  PROC DrawPart12()
    MoveL Offs(pOrigin,191.45,110.32,6.00),vTravel,z5,tPen\WObj:=wPaper;
    MoveL Offs(pOrigin,191.45,110.32,0.00),v60,z0,tPen\WObj:=wPaper;
    MoveL Offs(pOrigin,191.50,109.88,0.00),v40,z0,tPen\WObj:=wPaper;
    MoveL Offs(pOrigin,193.40,108.07,0.00),v40,fine,tPen\WObj:=wPaper;
    MoveL Offs(pOrigin,193.40,108.07,6.00),v60,z5,tPen\WObj:=wPaper;
    MoveL Offs(pOrigin,194.60,106.72,6.00),vTravel,z5,tPen\WObj:=wPaper;
    MoveL Offs(pOrigin,194.60,106.72,0.00),v60,z0,tPen\WObj:=wPaper;
    MoveL Offs(pOrigin,195.65,107.03,0.00),v40,z0,tPen\WObj:=wPaper;
    MoveL Offs(pOrigin,195.65,107.03,0.00),v40,z0,tPen\WObj:=wPaper;
    MoveL Offs(pOrigin,197.00,108.68,0.00),v40,z0,tPen\WObj:=wPaper;
    MoveL Offs(pOrigin,197.00,108.68,0.00),v40,z0,tPen\WObj:=wPaper;
    MoveL Offs(pOrigin,197.45,111.07,0.00),v40,z0,tPen\WObj:=wPaper;
    MoveL Offs(pOrigin,197.45,111.07,0.00),v40,z0,tPen\WObj:=wPaper;
    MoveL Offs(pOrigin,198.05,112.28,0.00),v40,z0,tPen\WObj:=wPaper;
    MoveL Offs(pOrigin,198.05,112.28,0.00),v40,z0,tPen\WObj:=wPaper;
    MoveL Offs(pOrigin,199.10,113.78,0.00),v40,z0,tPen\WObj:=wPaper;
    MoveL Offs(pOrigin,199.10,115.72,0.00),v40,z0,tPen\WObj:=wPaper;
    MoveL Offs(pOrigin,198.05,118.28,0.00),v40,z0,tPen\WObj:=wPaper;
    MoveL Offs(pOrigin,191.30,125.03,0.00),v40,z0,tPen\WObj:=wPaper;
    MoveL Offs(pOrigin,188.75,125.03,0.00),v40,fine,tPen\WObj:=wPaper;
    MoveL Offs(pOrigin,188.75,125.03,6.00),v60,z5,tPen\WObj:=wPaper;
    MoveL Offs(pOrigin,190.25,121.43,6.00),vTravel,z5,tPen\WObj:=wPaper;
    MoveL Offs(pOrigin,190.25,121.43,0.00),v60,z0,tPen\WObj:=wPaper;
    MoveL Offs(pOrigin,190.70,121.12,0.00),v40,z0,tPen\WObj:=wPaper;
    MoveL Offs(pOrigin,190.85,119.93,0.00),v40,z0,tPen\WObj:=wPaper;
    MoveL Offs(pOrigin,190.85,119.93,0.00),v40,z0,tPen\WObj:=wPaper;
    MoveL Offs(pOrigin,197.15,113.93,0.00),v40,z0,tPen\WObj:=wPaper;
    MoveL Offs(pOrigin,197.15,113.93,0.00),v40,z0,tPen\WObj:=wPaper;
    MoveL Offs(pOrigin,197.35,112.88,0.00),v40,z0,tPen\WObj:=wPaper;
    MoveL Offs(pOrigin,198.05,112.28,0.00),v40,fine,tPen\WObj:=wPaper;
    MoveL Offs(pOrigin,198.05,112.28,6.00),v60,z5,tPen\WObj:=wPaper;
    MoveL Offs(pOrigin,197.15,113.93,6.00),vTravel,z5,tPen\WObj:=wPaper;
    MoveL Offs(pOrigin,197.15,113.93,0.00),v60,z0,tPen\WObj:=wPaper;
    MoveL Offs(pOrigin,198.50,114.82,0.00),v40,fine,tPen\WObj:=wPaper;
    MoveL Offs(pOrigin,198.50,114.82,6.00),v60,z5,tPen\WObj:=wPaper;
    MoveL Offs(pOrigin,203.45,112.57,6.00),vTravel,z5,tPen\WObj:=wPaper;
    MoveL Offs(pOrigin,203.45,112.57,0.00),v60,z0,tPen\WObj:=wPaper;
    MoveL Offs(pOrigin,204.80,116.93,0.00),v40,fine,tPen\WObj:=wPaper;
    MoveL Offs(pOrigin,204.80,116.93,6.00),v60,z5,tPen\WObj:=wPaper;
    MoveL Offs(pOrigin,205.55,118.28,6.00),vTravel,z5,tPen\WObj:=wPaper;
    MoveL Offs(pOrigin,205.55,118.28,0.00),v60,z0,tPen\WObj:=wPaper;
    MoveL Offs(pOrigin,209.15,114.43,0.00),v40,z0,tPen\WObj:=wPaper;
    MoveL Offs(pOrigin,210.65,113.62,0.00),v40,z0,tPen\WObj:=wPaper;
    MoveL Offs(pOrigin,210.65,113.62,0.00),v40,z0,tPen\WObj:=wPaper;
    MoveL Offs(pOrigin,210.65,113.93,0.00),v40,z0,tPen\WObj:=wPaper;
    MoveL Offs(pOrigin,210.95,113.93,0.00),v40,z0,tPen\WObj:=wPaper;
    MoveL Offs(pOrigin,210.95,113.62,0.00),v40,z0,tPen\WObj:=wPaper;
    MoveL Offs(pOrigin,210.95,113.62,0.00),v40,z0,tPen\WObj:=wPaper;
    MoveL Offs(pOrigin,215.00,109.43,0.00),v40,z0,tPen\WObj:=wPaper;
    MoveL Offs(pOrigin,215.00,109.43,0.00),v40,z0,tPen\WObj:=wPaper;
    MoveL Offs(pOrigin,215.75,110.03,0.00),v40,z0,tPen\WObj:=wPaper;
    MoveL Offs(pOrigin,215.75,110.03,0.00),v40,z0,tPen\WObj:=wPaper;
    MoveL Offs(pOrigin,216.50,110.78,0.00),v40,z0,tPen\WObj:=wPaper;
    MoveL Offs(pOrigin,217.55,115.72,0.00),v40,z0,tPen\WObj:=wPaper;
    MoveL Offs(pOrigin,216.50,120.53,0.00),v40,z0,tPen\WObj:=wPaper;
    MoveL Offs(pOrigin,215.75,121.28,0.00),v40,z0,tPen\WObj:=wPaper;
    MoveL Offs(pOrigin,215.75,121.28,0.00),v40,z0,tPen\WObj:=wPaper;
    MoveL Offs(pOrigin,210.95,116.32,0.00),v40,z0,tPen\WObj:=wPaper;
    MoveL Offs(pOrigin,210.35,115.57,0.00),v40,z0,tPen\WObj:=wPaper;
    MoveL Offs(pOrigin,215.75,110.03,0.00),v40,z0,tPen\WObj:=wPaper;
    MoveL Offs(pOrigin,215.00,109.43,0.00),v40,z0,tPen\WObj:=wPaper;
    MoveL Offs(pOrigin,214.65,108.38,0.00),v40,z0,tPen\WObj:=wPaper;
    MoveL Offs(pOrigin,213.80,108.03,0.00),v40,z0,tPen\WObj:=wPaper;
    MoveL Offs(pOrigin,213.35,107.22,0.00),v40,z0,tPen\WObj:=wPaper;
    MoveL Offs(pOrigin,212.80,107.03,0.00),v40,z0,tPen\WObj:=wPaper;
    MoveL Offs(pOrigin,212.35,104.62,0.00),v40,z0,tPen\WObj:=wPaper;
    MoveL Offs(pOrigin,211.15,102.97,0.00),v40,z0,tPen\WObj:=wPaper;
    MoveL Offs(pOrigin,210.50,100.12,0.00),v40,z0,tPen\WObj:=wPaper;
    MoveL Offs(pOrigin,210.50,100.12,0.00),v40,z0,tPen\WObj:=wPaper;
    MoveL Offs(pOrigin,213.65,97.03,0.00),v40,z0,tPen\WObj:=wPaper;
    MoveL Offs(pOrigin,221.15,95.18,0.00),v40,z0,tPen\WObj:=wPaper;
    MoveL Offs(pOrigin,226.55,93.22,0.00),v40,fine,tPen\WObj:=wPaper;
    MoveL Offs(pOrigin,226.55,93.22,6.00),v60,z5,tPen\WObj:=wPaper;
    MoveL Offs(pOrigin,217.25,86.18,6.00),vTravel,z5,tPen\WObj:=wPaper;
    MoveL Offs(pOrigin,217.25,86.18,0.00),v60,z0,tPen\WObj:=wPaper;
    MoveL Offs(pOrigin,214.85,88.62,0.00),v40,z0,tPen\WObj:=wPaper;
    MoveL Offs(pOrigin,213.05,88.72,0.00),v40,z0,tPen\WObj:=wPaper;
    MoveL Offs(pOrigin,213.05,88.72,0.00),v40,z0,tPen\WObj:=wPaper;
    MoveL Offs(pOrigin,212.30,87.68,0.00),v40,z0,tPen\WObj:=wPaper;
    MoveL Offs(pOrigin,212.50,86.78,0.00),v40,z0,tPen\WObj:=wPaper;
    MoveL Offs(pOrigin,213.05,86.22,0.00),v40,z0,tPen\WObj:=wPaper;
    MoveL Offs(pOrigin,217.25,86.18,0.00),v40,z0,tPen\WObj:=wPaper;
    MoveL Offs(pOrigin,217.25,86.18,0.00),v40,z0,tPen\WObj:=wPaper;
    MoveL Offs(pOrigin,219.95,83.32,0.00),v40,z0,tPen\WObj:=wPaper;
    MoveL Offs(pOrigin,219.95,83.32,0.00),v40,z0,tPen\WObj:=wPaper;
    MoveL Offs(pOrigin,217.70,81.07,0.00),v40,z0,tPen\WObj:=wPaper;
    MoveL Offs(pOrigin,216.80,80.93,0.00),v40,z0,tPen\WObj:=wPaper;
    MoveL Offs(pOrigin,216.80,80.93,0.00),v40,z0,tPen\WObj:=wPaper;
    MoveL Offs(pOrigin,215.95,80.03,0.00),v40,z0,tPen\WObj:=wPaper;
    MoveL Offs(pOrigin,215.95,79.43,0.00),v40,z0,tPen\WObj:=wPaper;
    MoveL Offs(pOrigin,220.25,75.32,0.00),v40,z0,tPen\WObj:=wPaper;
    MoveL Offs(pOrigin,220.85,75.07,0.00),v40,z0,tPen\WObj:=wPaper;
    MoveL Offs(pOrigin,225.80,75.07,0.00),v40,z0,tPen\WObj:=wPaper;
    MoveL Offs(pOrigin,225.80,75.07,0.00),v40,z0,tPen\WObj:=wPaper;
    MoveL Offs(pOrigin,225.20,70.43,0.00),v40,z0,tPen\WObj:=wPaper;
    MoveL Offs(pOrigin,224.75,69.68,0.00),v40,z0,tPen\WObj:=wPaper;
    MoveL Offs(pOrigin,224.75,69.68,0.00),v40,z0,tPen\WObj:=wPaper;
    MoveL Offs(pOrigin,224.30,68.03,0.00),v40,z0,tPen\WObj:=wPaper;
    MoveL Offs(pOrigin,222.80,67.07,0.00),v40,z0,tPen\WObj:=wPaper;
    MoveL Offs(pOrigin,221.00,64.43,0.00),v40,z0,tPen\WObj:=wPaper;
    MoveL Offs(pOrigin,220.10,63.97,0.00),v40,z0,tPen\WObj:=wPaper;
    MoveL Offs(pOrigin,220.10,63.97,0.00),v40,z0,tPen\WObj:=wPaper;
    MoveL Offs(pOrigin,214.60,69.38,0.00),v40,z0,tPen\WObj:=wPaper;
    MoveL Offs(pOrigin,214.55,69.82,0.00),v40,z0,tPen\WObj:=wPaper;
    MoveL Offs(pOrigin,214.55,69.82,0.00),v40,z0,tPen\WObj:=wPaper;
    MoveL Offs(pOrigin,215.00,70.88,0.00),v40,z0,tPen\WObj:=wPaper;
    MoveL Offs(pOrigin,214.55,69.82,0.00),v40,z0,tPen\WObj:=wPaper;
    MoveL Offs(pOrigin,212.75,71.47,0.00),v40,fine,tPen\WObj:=wPaper;
    MoveL Offs(pOrigin,212.75,71.47,6.00),v60,z5,tPen\WObj:=wPaper;
    MoveL Offs(pOrigin,210.80,70.57,6.00),vTravel,z5,tPen\WObj:=wPaper;
    MoveL Offs(pOrigin,210.80,70.57,0.00),v60,z0,tPen\WObj:=wPaper;
    MoveL Offs(pOrigin,211.85,71.43,0.00),v40,z0,tPen\WObj:=wPaper;
    MoveL Offs(pOrigin,213.20,71.93,0.00),v40,z0,tPen\WObj:=wPaper;
    MoveL Offs(pOrigin,214.25,73.88,0.00),v40,z0,tPen\WObj:=wPaper;
    MoveL Offs(pOrigin,214.25,73.88,0.00),v40,z0,tPen\WObj:=wPaper;
    MoveL Offs(pOrigin,214.60,75.53,0.00),v40,z0,tPen\WObj:=wPaper;
    MoveL Offs(pOrigin,215.15,76.28,0.00),v40,z0,tPen\WObj:=wPaper;
    MoveL Offs(pOrigin,215.15,76.28,0.00),v40,z0,tPen\WObj:=wPaper;
    MoveL Offs(pOrigin,215.45,78.38,0.00),v40,z0,tPen\WObj:=wPaper;
    MoveL Offs(pOrigin,215.45,78.38,0.00),v40,z0,tPen\WObj:=wPaper;
  ENDPROC

  PROC DrawPart13()
    MoveL Offs(pOrigin,215.90,79.28,0.00),v40,fine,tPen\WObj:=wPaper;
    MoveL Offs(pOrigin,215.90,79.28,6.00),v60,z5,tPen\WObj:=wPaper;
    MoveL Offs(pOrigin,216.35,80.78,6.00),vTravel,z5,tPen\WObj:=wPaper;
    MoveL Offs(pOrigin,216.35,80.78,0.00),v60,z0,tPen\WObj:=wPaper;
    MoveL Offs(pOrigin,214.40,80.93,0.00),v40,z0,tPen\WObj:=wPaper;
    MoveL Offs(pOrigin,212.00,81.68,0.00),v40,z0,tPen\WObj:=wPaper;
    MoveL Offs(pOrigin,208.85,81.68,0.00),v40,z0,tPen\WObj:=wPaper;
    MoveL Offs(pOrigin,207.35,82.18,0.00),v40,z0,tPen\WObj:=wPaper;
    MoveL Offs(pOrigin,206.00,83.62,0.00),v40,z0,tPen\WObj:=wPaper;
    MoveL Offs(pOrigin,206.30,85.43,0.00),v40,z0,tPen\WObj:=wPaper;
    MoveL Offs(pOrigin,206.30,85.43,0.00),v40,z0,tPen\WObj:=wPaper;
    MoveL Offs(pOrigin,203.00,88.57,0.00),v40,z0,tPen\WObj:=wPaper;
    MoveL Offs(pOrigin,202.85,89.18,0.00),v40,z0,tPen\WObj:=wPaper;
    MoveL Offs(pOrigin,202.85,89.18,0.00),v40,z0,tPen\WObj:=wPaper;
    MoveL Offs(pOrigin,203.60,89.93,0.00),v40,z0,tPen\WObj:=wPaper;
    MoveL Offs(pOrigin,203.60,89.93,0.00),v40,z0,tPen\WObj:=wPaper;
    MoveL Offs(pOrigin,202.85,89.18,0.00),v40,z0,tPen\WObj:=wPaper;
    MoveL Offs(pOrigin,202.85,89.18,0.00),v40,z0,tPen\WObj:=wPaper;
    MoveL Offs(pOrigin,202.25,89.93,0.00),v40,fine,tPen\WObj:=wPaper;
    MoveL Offs(pOrigin,202.25,89.93,6.00),v60,z5,tPen\WObj:=wPaper;
    MoveL Offs(pOrigin,203.60,89.93,6.00),vTravel,z5,tPen\WObj:=wPaper;
    MoveL Offs(pOrigin,203.60,89.93,0.00),v60,z0,tPen\WObj:=wPaper;
    MoveL Offs(pOrigin,204.35,89.78,0.00),v40,z0,tPen\WObj:=wPaper;
    MoveL Offs(pOrigin,206.90,87.38,0.00),v40,z0,tPen\WObj:=wPaper;
    MoveL Offs(pOrigin,206.90,87.38,0.00),v40,z0,tPen\WObj:=wPaper;
    MoveL Offs(pOrigin,206.90,86.18,0.00),v40,z0,tPen\WObj:=wPaper;
    MoveL Offs(pOrigin,206.30,85.43,0.00),v40,fine,tPen\WObj:=wPaper;
    MoveL Offs(pOrigin,206.30,85.43,6.00),v60,z5,tPen\WObj:=wPaper;
    MoveL Offs(pOrigin,206.90,87.38,6.00),vTravel,z5,tPen\WObj:=wPaper;
    MoveL Offs(pOrigin,206.90,87.38,0.00),v60,z0,tPen\WObj:=wPaper;
    MoveL Offs(pOrigin,209.30,88.88,0.00),v40,z0,tPen\WObj:=wPaper;
    MoveL Offs(pOrigin,208.85,88.28,0.00),v40,z0,tPen\WObj:=wPaper;
    MoveL Offs(pOrigin,209.60,88.88,0.00),v40,z0,tPen\WObj:=wPaper;
    MoveL Offs(pOrigin,213.05,88.72,0.00),v40,z0,tPen\WObj:=wPaper;
    MoveL Offs(pOrigin,213.05,88.72,0.00),v40,z0,tPen\WObj:=wPaper;
    MoveL Offs(pOrigin,212.30,87.97,0.00),v40,fine,tPen\WObj:=wPaper;
    MoveL Offs(pOrigin,212.30,87.97,6.00),v60,z5,tPen\WObj:=wPaper;
    MoveL Offs(pOrigin,211.70,85.43,6.00),vTravel,z5,tPen\WObj:=wPaper;
    MoveL Offs(pOrigin,211.70,85.43,0.00),v60,z0,tPen\WObj:=wPaper;
    MoveL Offs(pOrigin,211.50,86.18,0.00),v40,z0,tPen\WObj:=wPaper;
    MoveL Offs(pOrigin,210.20,86.78,0.00),v40,z0,tPen\WObj:=wPaper;
    MoveL Offs(pOrigin,208.85,88.28,0.00),v40,fine,tPen\WObj:=wPaper;
    MoveL Offs(pOrigin,208.85,88.28,6.00),v60,z5,tPen\WObj:=wPaper;
    MoveL Offs(pOrigin,206.00,83.32,6.00),vTravel,z5,tPen\WObj:=wPaper;
    MoveL Offs(pOrigin,206.00,83.32,0.00),v60,z0,tPen\WObj:=wPaper;
    MoveL Offs(pOrigin,205.40,81.82,0.00),v40,z0,tPen\WObj:=wPaper;
    MoveL Offs(pOrigin,205.40,81.82,0.00),v40,z0,tPen\WObj:=wPaper;
    MoveL Offs(pOrigin,205.55,80.47,0.00),v40,z0,tPen\WObj:=wPaper;
    MoveL Offs(pOrigin,205.55,80.47,0.00),v40,z0,tPen\WObj:=wPaper;
    MoveL Offs(pOrigin,205.05,79.88,0.00),v40,z0,tPen\WObj:=wPaper;
    MoveL Offs(pOrigin,204.50,77.62,0.00),v40,z0,tPen\WObj:=wPaper;
    MoveL Offs(pOrigin,204.50,77.62,0.00),v40,z0,tPen\WObj:=wPaper;
    MoveL Offs(pOrigin,203.90,76.88,0.00),v40,z0,tPen\WObj:=wPaper;
    MoveL Offs(pOrigin,203.90,76.88,0.00),v40,z0,tPen\WObj:=wPaper;
    MoveL Offs(pOrigin,203.45,74.93,0.00),v40,z0,tPen\WObj:=wPaper;
    MoveL Offs(pOrigin,203.45,74.93,0.00),v40,z0,tPen\WObj:=wPaper;
    MoveL Offs(pOrigin,205.55,73.28,0.00),v40,z0,tPen\WObj:=wPaper;
    MoveL Offs(pOrigin,206.60,71.62,0.00),v40,z0,tPen\WObj:=wPaper;
    MoveL Offs(pOrigin,208.25,69.97,0.00),v40,z0,tPen\WObj:=wPaper;
    MoveL Offs(pOrigin,208.25,69.53,0.00),v40,z0,tPen\WObj:=wPaper;
    MoveL Offs(pOrigin,209.00,70.53,0.00),v40,z0,tPen\WObj:=wPaper;
    MoveL Offs(pOrigin,210.80,70.57,0.00),v40,z0,tPen\WObj:=wPaper;
    MoveL Offs(pOrigin,210.80,70.57,0.00),v40,z0,tPen\WObj:=wPaper;
    MoveL Offs(pOrigin,211.80,69.53,0.00),v40,z0,tPen\WObj:=wPaper;
    MoveL Offs(pOrigin,212.45,67.88,0.00),v40,z0,tPen\WObj:=wPaper;
    MoveL Offs(pOrigin,218.15,62.33,0.00),v40,z0,tPen\WObj:=wPaper;
    MoveL Offs(pOrigin,218.15,62.33,0.00),v40,z0,tPen\WObj:=wPaper;
    MoveL Offs(pOrigin,218.15,61.88,0.00),v40,z0,tPen\WObj:=wPaper;
    MoveL Offs(pOrigin,217.55,61.58,0.00),v40,z0,tPen\WObj:=wPaper;
    MoveL Offs(pOrigin,217.55,61.58,0.00),v40,z0,tPen\WObj:=wPaper;
    MoveL Offs(pOrigin,212.90,66.22,0.00),v40,z0,tPen\WObj:=wPaper;
    MoveL Offs(pOrigin,212.00,66.72,0.00),v40,z0,tPen\WObj:=wPaper;
    MoveL Offs(pOrigin,211.45,66.22,0.00),v40,z0,tPen\WObj:=wPaper;
    MoveL Offs(pOrigin,211.85,65.47,0.00),v40,z0,tPen\WObj:=wPaper;
    MoveL Offs(pOrigin,212.15,65.18,0.00),v40,z0,tPen\WObj:=wPaper;
    MoveL Offs(pOrigin,216.80,60.53,0.00),v40,z0,tPen\WObj:=wPaper;
    MoveL Offs(pOrigin,216.80,60.53,0.00),v40,z0,tPen\WObj:=wPaper;
    MoveL Offs(pOrigin,217.55,61.58,0.00),v40,z0,tPen\WObj:=wPaper;
    MoveL Offs(pOrigin,218.15,62.33,0.00),v40,z0,tPen\WObj:=wPaper;
    MoveL Offs(pOrigin,219.35,62.78,0.00),v40,z0,tPen\WObj:=wPaper;
    MoveL Offs(pOrigin,220.10,63.97,0.00),v40,fine,tPen\WObj:=wPaper;
    MoveL Offs(pOrigin,220.10,63.97,6.00),v60,z5,tPen\WObj:=wPaper;
    MoveL Offs(pOrigin,221.90,65.93,6.00),vTravel,z5,tPen\WObj:=wPaper;
    MoveL Offs(pOrigin,221.90,65.93,0.00),v60,z0,tPen\WObj:=wPaper;
    MoveL Offs(pOrigin,214.25,73.57,0.00),v40,z0,tPen\WObj:=wPaper;
    MoveL Offs(pOrigin,213.35,73.88,0.00),v40,z0,tPen\WObj:=wPaper;
    MoveL Offs(pOrigin,213.05,73.72,0.00),v40,z0,tPen\WObj:=wPaper;
    MoveL Offs(pOrigin,213.05,74.03,0.00),v40,z0,tPen\WObj:=wPaper;
    MoveL Offs(pOrigin,213.35,73.88,0.00),v40,z0,tPen\WObj:=wPaper;
    MoveL Offs(pOrigin,213.05,73.72,0.00),v40,z0,tPen\WObj:=wPaper;
    MoveL Offs(pOrigin,213.05,74.03,0.00),v40,z0,tPen\WObj:=wPaper;
    MoveL Offs(pOrigin,213.35,73.88,0.00),v40,fine,tPen\WObj:=wPaper;
    MoveL Offs(pOrigin,213.35,73.88,6.00),v60,z5,tPen\WObj:=wPaper;
    MoveL Offs(pOrigin,213.50,76.72,6.00),vTravel,z5,tPen\WObj:=wPaper;
    MoveL Offs(pOrigin,213.50,76.72,0.00),v60,z0,tPen\WObj:=wPaper;
    MoveL Offs(pOrigin,215.00,78.22,0.00),v40,z0,tPen\WObj:=wPaper;
    MoveL Offs(pOrigin,213.50,76.72,0.00),v40,fine,tPen\WObj:=wPaper;
    MoveL Offs(pOrigin,213.50,76.72,6.00),v60,z5,tPen\WObj:=wPaper;
    MoveL Offs(pOrigin,215.15,76.28,6.00),vTravel,z5,tPen\WObj:=wPaper;
    MoveL Offs(pOrigin,215.15,76.28,0.00),v60,z0,tPen\WObj:=wPaper;
    MoveL Offs(pOrigin,218.30,73.43,0.00),v40,z0,tPen\WObj:=wPaper;
    MoveL Offs(pOrigin,219.35,71.78,0.00),v40,z0,tPen\WObj:=wPaper;
    MoveL Offs(pOrigin,223.40,67.72,0.00),v40,fine,tPen\WObj:=wPaper;
    MoveL Offs(pOrigin,223.40,67.72,6.00),v60,z5,tPen\WObj:=wPaper;
    MoveL Offs(pOrigin,224.75,69.68,6.00),vTravel,z5,tPen\WObj:=wPaper;
    MoveL Offs(pOrigin,224.75,69.68,0.00),v60,z0,tPen\WObj:=wPaper;
    MoveL Offs(pOrigin,221.00,73.43,0.00),v40,z0,tPen\WObj:=wPaper;
    MoveL Offs(pOrigin,220.10,73.57,0.00),v40,z0,tPen\WObj:=wPaper;
    MoveL Offs(pOrigin,219.95,73.88,0.00),v40,z0,tPen\WObj:=wPaper;
    MoveL Offs(pOrigin,220.10,74.03,0.00),v40,z0,tPen\WObj:=wPaper;
    MoveL Offs(pOrigin,220.40,74.03,0.00),v40,z0,tPen\WObj:=wPaper;
    MoveL Offs(pOrigin,220.40,73.72,0.00),v40,z0,tPen\WObj:=wPaper;
    MoveL Offs(pOrigin,220.10,74.03,0.00),v40,z0,tPen\WObj:=wPaper;
    MoveL Offs(pOrigin,220.40,74.03,0.00),v40,z0,tPen\WObj:=wPaper;
    MoveL Offs(pOrigin,220.25,73.72,0.00),v40,z0,tPen\WObj:=wPaper;
    MoveL Offs(pOrigin,220.10,74.03,0.00),v40,fine,tPen\WObj:=wPaper;
    MoveL Offs(pOrigin,220.10,74.03,6.00),v60,z5,tPen\WObj:=wPaper;
    MoveL Offs(pOrigin,225.80,75.07,6.00),vTravel,z5,tPen\WObj:=wPaper;
    MoveL Offs(pOrigin,225.80,75.07,0.00),v60,z0,tPen\WObj:=wPaper;
    MoveL Offs(pOrigin,226.25,77.78,0.00),v40,z0,tPen\WObj:=wPaper;
  ENDPROC

  PROC DrawPart14()
    MoveL Offs(pOrigin,225.95,80.32,0.00),v40,z0,tPen\WObj:=wPaper;
    MoveL Offs(pOrigin,225.35,81.78,0.00),v40,z0,tPen\WObj:=wPaper;
    MoveL Offs(pOrigin,222.20,83.32,0.00),v40,z0,tPen\WObj:=wPaper;
    MoveL Offs(pOrigin,220.25,83.32,0.00),v40,z0,tPen\WObj:=wPaper;
    MoveL Offs(pOrigin,217.70,80.93,0.00),v40,fine,tPen\WObj:=wPaper;
    MoveL Offs(pOrigin,217.70,80.93,6.00),v60,z5,tPen\WObj:=wPaper;
    MoveL Offs(pOrigin,209.75,78.53,6.00),vTravel,z5,tPen\WObj:=wPaper;
    MoveL Offs(pOrigin,209.75,78.53,0.00),v60,z0,tPen\WObj:=wPaper;
    MoveL Offs(pOrigin,210.20,78.22,0.00),v40,z0,tPen\WObj:=wPaper;
    MoveL Offs(pOrigin,210.05,77.78,0.00),v40,z0,tPen\WObj:=wPaper;
    MoveL Offs(pOrigin,209.75,77.93,0.00),v40,fine,tPen\WObj:=wPaper;
    MoveL Offs(pOrigin,209.75,77.93,6.00),v60,z5,tPen\WObj:=wPaper;
    MoveL Offs(pOrigin,209.90,75.53,6.00),vTravel,z5,tPen\WObj:=wPaper;
    MoveL Offs(pOrigin,209.90,75.53,0.00),v60,z0,tPen\WObj:=wPaper;
    MoveL Offs(pOrigin,208.70,75.53,0.00),v40,z0,tPen\WObj:=wPaper;
    MoveL Offs(pOrigin,207.95,75.97,0.00),v40,fine,tPen\WObj:=wPaper;
    MoveL Offs(pOrigin,207.95,75.97,6.00),v60,z5,tPen\WObj:=wPaper;
    MoveL Offs(pOrigin,207.95,74.62,6.00),vTravel,z5,tPen\WObj:=wPaper;
    MoveL Offs(pOrigin,207.95,74.62,0.00),v60,z0,tPen\WObj:=wPaper;
    MoveL Offs(pOrigin,207.95,74.18,0.00),v40,z0,tPen\WObj:=wPaper;
    MoveL Offs(pOrigin,208.70,73.88,0.00),v40,z0,tPen\WObj:=wPaper;
    MoveL Offs(pOrigin,208.70,73.88,0.00),v40,z0,tPen\WObj:=wPaper;
    MoveL Offs(pOrigin,209.55,74.32,0.00),v40,z0,tPen\WObj:=wPaper;
    MoveL Offs(pOrigin,209.90,75.53,0.00),v40,fine,tPen\WObj:=wPaper;
    MoveL Offs(pOrigin,209.90,75.53,6.00),v60,z5,tPen\WObj:=wPaper;
    MoveL Offs(pOrigin,209.60,74.18,6.00),vTravel,z5,tPen\WObj:=wPaper;
    MoveL Offs(pOrigin,209.60,74.18,0.00),v60,z0,tPen\WObj:=wPaper;
    MoveL Offs(pOrigin,209.45,73.57,0.00),v40,z0,tPen\WObj:=wPaper;
    MoveL Offs(pOrigin,208.85,73.57,0.00),v40,z0,tPen\WObj:=wPaper;
    MoveL Offs(pOrigin,208.70,73.88,0.00),v40,z0,tPen\WObj:=wPaper;
    MoveL Offs(pOrigin,208.70,73.57,0.00),v40,z0,tPen\WObj:=wPaper;
    MoveL Offs(pOrigin,208.85,70.57,0.00),v40,fine,tPen\WObj:=wPaper;
    MoveL Offs(pOrigin,208.85,70.57,6.00),v60,z5,tPen\WObj:=wPaper;
    MoveL Offs(pOrigin,208.25,69.53,6.00),vTravel,z5,tPen\WObj:=wPaper;
    MoveL Offs(pOrigin,208.25,69.53,0.00),v60,z0,tPen\WObj:=wPaper;
    MoveL Offs(pOrigin,209.60,68.03,0.00),v40,z0,tPen\WObj:=wPaper;
    MoveL Offs(pOrigin,211.25,67.62,0.00),v40,z0,tPen\WObj:=wPaper;
    MoveL Offs(pOrigin,211.70,66.97,0.00),v40,fine,tPen\WObj:=wPaper;
    MoveL Offs(pOrigin,211.70,66.97,6.00),v60,z5,tPen\WObj:=wPaper;
    MoveL Offs(pOrigin,213.95,68.18,6.00),vTravel,z5,tPen\WObj:=wPaper;
    MoveL Offs(pOrigin,213.95,68.18,0.00),v60,z0,tPen\WObj:=wPaper;
    MoveL Offs(pOrigin,214.55,69.22,0.00),v40,fine,tPen\WObj:=wPaper;
    MoveL Offs(pOrigin,214.55,69.22,6.00),v60,z5,tPen\WObj:=wPaper;
    MoveL Offs(pOrigin,208.25,69.53,6.00),vTravel,z5,tPen\WObj:=wPaper;
    MoveL Offs(pOrigin,208.25,69.53,0.00),v60,z0,tPen\WObj:=wPaper;
    MoveL Offs(pOrigin,207.55,69.22,0.00),v40,z0,tPen\WObj:=wPaper;
    MoveL Offs(pOrigin,206.50,65.62,0.00),v40,z0,tPen\WObj:=wPaper;
    MoveL Offs(pOrigin,206.00,64.88,0.00),v40,z0,tPen\WObj:=wPaper;
    MoveL Offs(pOrigin,206.00,62.17,0.00),v40,z0,tPen\WObj:=wPaper;
    MoveL Offs(pOrigin,206.75,60.38,0.00),v40,z0,tPen\WObj:=wPaper;
    MoveL Offs(pOrigin,208.55,58.58,0.00),v40,z0,tPen\WObj:=wPaper;
    MoveL Offs(pOrigin,208.40,58.28,0.00),v40,z0,tPen\WObj:=wPaper;
    MoveL Offs(pOrigin,209.15,58.72,0.00),v40,z0,tPen\WObj:=wPaper;
    MoveL Offs(pOrigin,216.05,60.08,0.00),v40,z0,tPen\WObj:=wPaper;
    MoveL Offs(pOrigin,216.80,60.53,0.00),v40,fine,tPen\WObj:=wPaper;
    MoveL Offs(pOrigin,216.80,60.53,6.00),v60,z5,tPen\WObj:=wPaper;
    MoveL Offs(pOrigin,207.20,56.33,6.00),vTravel,z5,tPen\WObj:=wPaper;
    MoveL Offs(pOrigin,207.20,56.33,0.00),v60,z0,tPen\WObj:=wPaper;
    MoveL Offs(pOrigin,207.50,56.78,0.00),v40,z0,tPen\WObj:=wPaper;
    MoveL Offs(pOrigin,207.20,56.33,0.00),v40,fine,tPen\WObj:=wPaper;
    MoveL Offs(pOrigin,207.20,56.33,6.00),v60,z5,tPen\WObj:=wPaper;
    MoveL Offs(pOrigin,207.05,68.03,6.00),vTravel,z5,tPen\WObj:=wPaper;
    MoveL Offs(pOrigin,207.05,68.03,0.00),v60,z0,tPen\WObj:=wPaper;
    MoveL Offs(pOrigin,202.65,72.38,0.00),v40,z0,tPen\WObj:=wPaper;
    MoveL Offs(pOrigin,202.55,73.28,0.00),v40,z0,tPen\WObj:=wPaper;
    MoveL Offs(pOrigin,203.45,74.93,0.00),v40,fine,tPen\WObj:=wPaper;
    MoveL Offs(pOrigin,203.45,74.93,6.00),v60,z5,tPen\WObj:=wPaper;
    MoveL Offs(pOrigin,203.90,76.88,6.00),vTravel,z5,tPen\WObj:=wPaper;
    MoveL Offs(pOrigin,203.90,76.88,0.00),v60,z0,tPen\WObj:=wPaper;
    MoveL Offs(pOrigin,202.25,78.53,0.00),v40,z0,tPen\WObj:=wPaper;
    MoveL Offs(pOrigin,205.40,81.82,0.00),v40,z0,tPen\WObj:=wPaper;
    MoveL Offs(pOrigin,205.40,81.82,0.00),v40,z0,tPen\WObj:=wPaper;
    MoveL Offs(pOrigin,202.25,78.82,0.00),v40,fine,tPen\WObj:=wPaper;
    MoveL Offs(pOrigin,202.25,78.82,6.00),v60,z5,tPen\WObj:=wPaper;
    MoveL Offs(pOrigin,198.50,77.32,6.00),vTravel,z5,tPen\WObj:=wPaper;
    MoveL Offs(pOrigin,198.50,77.32,0.00),v60,z0,tPen\WObj:=wPaper;
    MoveL Offs(pOrigin,197.15,76.43,0.00),v40,z0,tPen\WObj:=wPaper;
    MoveL Offs(pOrigin,197.15,76.43,0.00),v40,z0,tPen\WObj:=wPaper;
    MoveL Offs(pOrigin,197.30,74.47,0.00),v40,z0,tPen\WObj:=wPaper;
    MoveL Offs(pOrigin,197.60,74.32,0.00),v40,z0,tPen\WObj:=wPaper;
    MoveL Offs(pOrigin,197.60,73.12,0.00),v40,z0,tPen\WObj:=wPaper;
    MoveL Offs(pOrigin,197.15,72.38,0.00),v40,z0,tPen\WObj:=wPaper;
    MoveL Offs(pOrigin,197.15,72.38,0.00),v40,z0,tPen\WObj:=wPaper;
    MoveL Offs(pOrigin,197.05,71.47,0.00),v40,z0,tPen\WObj:=wPaper;
    MoveL Offs(pOrigin,195.50,69.57,0.00),v40,z0,tPen\WObj:=wPaper;
    MoveL Offs(pOrigin,194.60,69.38,0.00),v40,z0,tPen\WObj:=wPaper;
    MoveL Offs(pOrigin,194.60,69.38,0.00),v40,z0,tPen\WObj:=wPaper;
    MoveL Offs(pOrigin,193.60,65.62,0.00),v40,z0,tPen\WObj:=wPaper;
    MoveL Offs(pOrigin,191.75,61.12,0.00),v40,z0,tPen\WObj:=wPaper;
    MoveL Offs(pOrigin,191.90,60.03,0.00),v40,z0,tPen\WObj:=wPaper;
    MoveL Offs(pOrigin,198.90,66.68,0.00),v40,z0,tPen\WObj:=wPaper;
    MoveL Offs(pOrigin,198.60,67.53,0.00),v40,z0,tPen\WObj:=wPaper;
    MoveL Offs(pOrigin,197.15,68.03,0.00),v40,z0,tPen\WObj:=wPaper;
    MoveL Offs(pOrigin,195.65,69.53,0.00),v40,z0,tPen\WObj:=wPaper;
    MoveL Offs(pOrigin,194.60,69.38,0.00),v40,z0,tPen\WObj:=wPaper;
    MoveL Offs(pOrigin,193.40,70.88,0.00),v40,fine,tPen\WObj:=wPaper;
    MoveL Offs(pOrigin,193.40,70.88,6.00),v60,z5,tPen\WObj:=wPaper;
    MoveL Offs(pOrigin,192.95,72.97,6.00),vTravel,z5,tPen\WObj:=wPaper;
    MoveL Offs(pOrigin,192.95,72.97,0.00),v60,z0,tPen\WObj:=wPaper;
    MoveL Offs(pOrigin,193.40,72.38,0.00),v40,z0,tPen\WObj:=wPaper;
    MoveL Offs(pOrigin,193.25,70.97,0.00),v40,z0,tPen\WObj:=wPaper;
    MoveL Offs(pOrigin,191.45,72.82,0.00),v40,fine,tPen\WObj:=wPaper;
    MoveL Offs(pOrigin,191.45,72.82,6.00),v60,z5,tPen\WObj:=wPaper;
    MoveL Offs(pOrigin,188.75,69.97,6.00),vTravel,z5,tPen\WObj:=wPaper;
    MoveL Offs(pOrigin,188.75,69.97,0.00),v60,z0,tPen\WObj:=wPaper;
    MoveL Offs(pOrigin,189.50,68.62,0.00),v40,z0,tPen\WObj:=wPaper;
    MoveL Offs(pOrigin,193.10,65.18,0.00),v40,fine,tPen\WObj:=wPaper;
    MoveL Offs(pOrigin,193.10,65.18,6.00),v60,z5,tPen\WObj:=wPaper;
    MoveL Offs(pOrigin,192.20,62.62,6.00),vTravel,z5,tPen\WObj:=wPaper;
    MoveL Offs(pOrigin,192.20,62.62,0.00),v60,z0,tPen\WObj:=wPaper;
    MoveL Offs(pOrigin,186.65,67.88,0.00),v40,z0,tPen\WObj:=wPaper;
    MoveL Offs(pOrigin,185.90,69.38,0.00),v40,z0,tPen\WObj:=wPaper;
    MoveL Offs(pOrigin,182.90,72.38,0.00),v40,fine,tPen\WObj:=wPaper;
    MoveL Offs(pOrigin,182.90,72.38,6.00),v60,z5,tPen\WObj:=wPaper;
    MoveL Offs(pOrigin,182.30,74.32,6.00),vTravel,z5,tPen\WObj:=wPaper;
    MoveL Offs(pOrigin,182.30,74.32,0.00),v60,z0,tPen\WObj:=wPaper;
    MoveL Offs(pOrigin,184.10,76.12,0.00),v40,z0,tPen\WObj:=wPaper;
    MoveL Offs(pOrigin,182.30,74.32,0.00),v40,fine,tPen\WObj:=wPaper;
    MoveL Offs(pOrigin,182.30,74.32,6.00),v60,z5,tPen\WObj:=wPaper;
    MoveL Offs(pOrigin,180.95,72.97,6.00),vTravel,z5,tPen\WObj:=wPaper;
  ENDPROC

  PROC DrawPart15()
    MoveL Offs(pOrigin,180.95,72.97,0.00),v60,z0,tPen\WObj:=wPaper;
    MoveL Offs(pOrigin,182.00,74.03,0.00),v40,z0,tPen\WObj:=wPaper;
    MoveL Offs(pOrigin,180.95,72.97,0.00),v40,z0,tPen\WObj:=wPaper;
    MoveL Offs(pOrigin,180.65,72.38,0.00),v40,z0,tPen\WObj:=wPaper;
    MoveL Offs(pOrigin,179.75,71.62,0.00),v40,z0,tPen\WObj:=wPaper;
    MoveL Offs(pOrigin,179.75,71.62,0.00),v40,z0,tPen\WObj:=wPaper;
    MoveL Offs(pOrigin,179.30,72.22,0.00),v40,z0,tPen\WObj:=wPaper;
    MoveL Offs(pOrigin,179.30,77.62,0.00),v40,z0,tPen\WObj:=wPaper;
    MoveL Offs(pOrigin,179.30,77.62,0.00),v40,z0,tPen\WObj:=wPaper;
    MoveL Offs(pOrigin,179.35,84.22,0.00),v40,z0,tPen\WObj:=wPaper;
    MoveL Offs(pOrigin,179.90,84.78,0.00),v40,z0,tPen\WObj:=wPaper;
    MoveL Offs(pOrigin,181.55,84.97,0.00),v40,z0,tPen\WObj:=wPaper;
    MoveL Offs(pOrigin,185.30,88.68,0.00),v40,z0,tPen\WObj:=wPaper;
    MoveL Offs(pOrigin,186.20,88.78,0.00),v40,z0,tPen\WObj:=wPaper;
    MoveL Offs(pOrigin,186.95,89.32,0.00),v40,z0,tPen\WObj:=wPaper;
    MoveL Offs(pOrigin,188.60,89.47,0.00),v40,z0,tPen\WObj:=wPaper;
    MoveL Offs(pOrigin,189.65,89.18,0.00),v40,z0,tPen\WObj:=wPaper;
    MoveL Offs(pOrigin,190.40,89.72,0.00),v40,z0,tPen\WObj:=wPaper;
    MoveL Offs(pOrigin,191.15,89.78,0.00),v40,z0,tPen\WObj:=wPaper;
    MoveL Offs(pOrigin,194.00,87.07,0.00),v40,z0,tPen\WObj:=wPaper;
    MoveL Offs(pOrigin,194.00,87.07,0.00),v40,z0,tPen\WObj:=wPaper;
    MoveL Offs(pOrigin,194.00,86.03,0.00),v40,z0,tPen\WObj:=wPaper;
    MoveL Offs(pOrigin,193.55,85.57,0.00),v40,z0,tPen\WObj:=wPaper;
    MoveL Offs(pOrigin,193.55,85.57,0.00),v40,z0,tPen\WObj:=wPaper;
    MoveL Offs(pOrigin,193.55,84.53,0.00),v40,z0,tPen\WObj:=wPaper;
    MoveL Offs(pOrigin,193.10,83.78,0.00),v40,z0,tPen\WObj:=wPaper;
    MoveL Offs(pOrigin,193.10,83.78,0.00),v40,z0,tPen\WObj:=wPaper;
    MoveL Offs(pOrigin,194.60,82.12,0.00),v40,z0,tPen\WObj:=wPaper;
    MoveL Offs(pOrigin,195.35,81.97,0.00),v40,z0,tPen\WObj:=wPaper;
    MoveL Offs(pOrigin,195.35,81.97,0.00),v40,z0,tPen\WObj:=wPaper;
    MoveL Offs(pOrigin,198.20,84.97,0.00),v40,z0,tPen\WObj:=wPaper;
    MoveL Offs(pOrigin,198.20,84.97,0.00),v40,z0,tPen\WObj:=wPaper;
    MoveL Offs(pOrigin,198.80,85.43,0.00),v40,z0,tPen\WObj:=wPaper;
    MoveL Offs(pOrigin,198.65,86.62,0.00),v40,z0,tPen\WObj:=wPaper;
    MoveL Offs(pOrigin,197.00,88.22,0.00),v40,z0,tPen\WObj:=wPaper;
    MoveL Offs(pOrigin,195.95,88.28,0.00),v40,z0,tPen\WObj:=wPaper;
    MoveL Offs(pOrigin,195.50,87.97,0.00),v40,z0,tPen\WObj:=wPaper;
    MoveL Offs(pOrigin,195.50,87.97,0.00),v40,z0,tPen\WObj:=wPaper;
    MoveL Offs(pOrigin,198.20,84.97,0.00),v40,z0,tPen\WObj:=wPaper;
    MoveL Offs(pOrigin,198.20,84.97,0.00),v40,z0,tPen\WObj:=wPaper;
    MoveL Offs(pOrigin,195.35,81.97,0.00),v40,z0,tPen\WObj:=wPaper;
    MoveL Offs(pOrigin,195.35,81.97,0.00),v40,z0,tPen\WObj:=wPaper;
    MoveL Offs(pOrigin,196.40,81.53,0.00),v40,z0,tPen\WObj:=wPaper;
    MoveL Offs(pOrigin,197.15,81.57,0.00),v40,z0,tPen\WObj:=wPaper;
    MoveL Offs(pOrigin,198.80,83.18,0.00),v40,fine,tPen\WObj:=wPaper;
    MoveL Offs(pOrigin,198.80,83.18,6.00),v60,z5,tPen\WObj:=wPaper;
    MoveL Offs(pOrigin,198.65,84.97,6.00),vTravel,z5,tPen\WObj:=wPaper;
    MoveL Offs(pOrigin,198.65,84.97,0.00),v60,z0,tPen\WObj:=wPaper;
    MoveL Offs(pOrigin,199.10,84.07,0.00),v40,z0,tPen\WObj:=wPaper;
    MoveL Offs(pOrigin,199.00,83.32,0.00),v40,z0,tPen\WObj:=wPaper;
    MoveL Offs(pOrigin,197.30,81.53,0.00),v40,z0,tPen\WObj:=wPaper;
    MoveL Offs(pOrigin,197.30,81.53,0.00),v40,z0,tPen\WObj:=wPaper;
    MoveL Offs(pOrigin,198.30,80.47,0.00),v40,z0,tPen\WObj:=wPaper;
    MoveL Offs(pOrigin,199.10,78.38,0.00),v40,z0,tPen\WObj:=wPaper;
    MoveL Offs(pOrigin,198.85,75.68,0.00),v40,z0,tPen\WObj:=wPaper;
    MoveL Offs(pOrigin,197.60,74.32,0.00),v40,z0,tPen\WObj:=wPaper;
    MoveL Offs(pOrigin,197.60,74.32,0.00),v40,z0,tPen\WObj:=wPaper;
    MoveL Offs(pOrigin,198.50,75.22,0.00),v40,fine,tPen\WObj:=wPaper;
    MoveL Offs(pOrigin,198.50,75.22,6.00),v60,z5,tPen\WObj:=wPaper;
    MoveL Offs(pOrigin,197.15,76.43,6.00),vTravel,z5,tPen\WObj:=wPaper;
    MoveL Offs(pOrigin,197.15,76.43,0.00),v60,z0,tPen\WObj:=wPaper;
    MoveL Offs(pOrigin,191.30,82.12,0.00),v40,z0,tPen\WObj:=wPaper;
    MoveL Offs(pOrigin,190.40,82.12,0.00),v40,z0,tPen\WObj:=wPaper;
    MoveL Offs(pOrigin,191.30,82.28,0.00),v40,z0,tPen\WObj:=wPaper;
    MoveL Offs(pOrigin,191.75,83.47,0.00),v40,z0,tPen\WObj:=wPaper;
    MoveL Offs(pOrigin,191.75,83.47,0.00),v40,z0,tPen\WObj:=wPaper;
    MoveL Offs(pOrigin,189.05,86.18,0.00),v40,z0,tPen\WObj:=wPaper;
    MoveL Offs(pOrigin,189.05,86.18,0.00),v40,z0,tPen\WObj:=wPaper;
    MoveL Offs(pOrigin,188.75,88.57,0.00),v40,z0,tPen\WObj:=wPaper;
    MoveL Offs(pOrigin,188.30,89.32,0.00),v40,fine,tPen\WObj:=wPaper;
    MoveL Offs(pOrigin,188.30,89.32,6.00),v60,z5,tPen\WObj:=wPaper;
    MoveL Offs(pOrigin,189.95,89.18,6.00),vTravel,z5,tPen\WObj:=wPaper;
    MoveL Offs(pOrigin,189.95,89.18,0.00),v60,z0,tPen\WObj:=wPaper;
    MoveL Offs(pOrigin,190.00,88.78,0.00),v40,z0,tPen\WObj:=wPaper;
    MoveL Offs(pOrigin,193.55,85.57,0.00),v40,fine,tPen\WObj:=wPaper;
    MoveL Offs(pOrigin,193.55,85.57,6.00),v60,z5,tPen\WObj:=wPaper;
    MoveL Offs(pOrigin,194.00,87.07,6.00),vTravel,z5,tPen\WObj:=wPaper;
    MoveL Offs(pOrigin,194.00,87.07,0.00),v60,z0,tPen\WObj:=wPaper;
    MoveL Offs(pOrigin,194.75,87.93,0.00),v40,z0,tPen\WObj:=wPaper;
    MoveL Offs(pOrigin,195.50,87.97,0.00),v40,fine,tPen\WObj:=wPaper;
    MoveL Offs(pOrigin,195.50,87.97,6.00),v60,z5,tPen\WObj:=wPaper;
    MoveL Offs(pOrigin,193.10,83.78,6.00),vTravel,z5,tPen\WObj:=wPaper;
    MoveL Offs(pOrigin,193.10,83.78,0.00),v60,z0,tPen\WObj:=wPaper;
    MoveL Offs(pOrigin,191.75,83.47,0.00),v40,fine,tPen\WObj:=wPaper;
    MoveL Offs(pOrigin,191.75,83.47,6.00),v60,z5,tPen\WObj:=wPaper;
    MoveL Offs(pOrigin,190.40,82.12,6.00),vTravel,z5,tPen\WObj:=wPaper;
    MoveL Offs(pOrigin,190.40,82.12,0.00),v60,z0,tPen\WObj:=wPaper;
    MoveL Offs(pOrigin,189.05,82.68,0.00),v40,z0,tPen\WObj:=wPaper;
    MoveL Offs(pOrigin,185.15,78.82,0.00),v40,fine,tPen\WObj:=wPaper;
    MoveL Offs(pOrigin,185.15,78.82,6.00),v60,z5,tPen\WObj:=wPaper;
    MoveL Offs(pOrigin,184.10,77.93,6.00),vTravel,z5,tPen\WObj:=wPaper;
    MoveL Offs(pOrigin,184.10,77.93,0.00),v60,z0,tPen\WObj:=wPaper;
    MoveL Offs(pOrigin,184.85,77.32,0.00),v40,z0,tPen\WObj:=wPaper;
    MoveL Offs(pOrigin,185.00,77.03,0.00),v40,z0,tPen\WObj:=wPaper;
    MoveL Offs(pOrigin,180.80,72.43,0.00),v40,z0,tPen\WObj:=wPaper;
    MoveL Offs(pOrigin,182.60,72.38,0.00),v40,z0,tPen\WObj:=wPaper;
    MoveL Offs(pOrigin,184.10,72.97,0.00),v40,z0,tPen\WObj:=wPaper;
    MoveL Offs(pOrigin,185.15,73.03,0.00),v40,z0,tPen\WObj:=wPaper;
    MoveL Offs(pOrigin,185.90,73.62,0.00),v40,z0,tPen\WObj:=wPaper;
    MoveL Offs(pOrigin,187.55,74.07,0.00),v40,z0,tPen\WObj:=wPaper;
    MoveL Offs(pOrigin,189.00,76.72,0.00),v40,z0,tPen\WObj:=wPaper;
    MoveL Offs(pOrigin,189.45,78.82,0.00),v40,z0,tPen\WObj:=wPaper;
    MoveL Offs(pOrigin,189.95,79.43,0.00),v40,fine,tPen\WObj:=wPaper;
    MoveL Offs(pOrigin,189.95,79.43,6.00),v60,z5,tPen\WObj:=wPaper;
    MoveL Offs(pOrigin,188.90,82.72,6.00),vTravel,z5,tPen\WObj:=wPaper;
    MoveL Offs(pOrigin,188.90,82.72,0.00),v60,z0,tPen\WObj:=wPaper;
    MoveL Offs(pOrigin,184.85,78.57,0.00),v40,z0,tPen\WObj:=wPaper;
    MoveL Offs(pOrigin,183.35,77.62,0.00),v40,z0,tPen\WObj:=wPaper;
    MoveL Offs(pOrigin,183.35,77.62,0.00),v40,z0,tPen\WObj:=wPaper;
    MoveL Offs(pOrigin,179.30,77.62,0.00),v40,fine,tPen\WObj:=wPaper;
    MoveL Offs(pOrigin,179.30,77.62,6.00),v60,z5,tPen\WObj:=wPaper;
    MoveL Offs(pOrigin,180.65,72.38,6.00),vTravel,z5,tPen\WObj:=wPaper;
    MoveL Offs(pOrigin,180.65,72.38,0.00),v60,z0,tPen\WObj:=wPaper;
    MoveL Offs(pOrigin,179.75,71.62,0.00),v40,z0,tPen\WObj:=wPaper;
    MoveL Offs(pOrigin,179.75,71.62,0.00),v40,z0,tPen\WObj:=wPaper;
    MoveL Offs(pOrigin,179.75,63.38,0.00),v40,z0,tPen\WObj:=wPaper;
    MoveL Offs(pOrigin,180.35,61.58,0.00),v40,z0,tPen\WObj:=wPaper;
    MoveL Offs(pOrigin,180.35,61.58,0.00),v40,z0,tPen\WObj:=wPaper;
    MoveL Offs(pOrigin,180.40,59.78,0.00),v40,z0,tPen\WObj:=wPaper;
    MoveL Offs(pOrigin,182.00,58.28,0.00),v40,z0,tPen\WObj:=wPaper;
  ENDPROC

  PROC DrawPart16()
    MoveL Offs(pOrigin,190.25,58.28,0.00),v40,z0,tPen\WObj:=wPaper;
    MoveL Offs(pOrigin,190.25,58.28,0.00),v40,z0,tPen\WObj:=wPaper;
    MoveL Offs(pOrigin,191.75,59.92,0.00),v40,z0,tPen\WObj:=wPaper;
    MoveL Offs(pOrigin,191.75,59.92,0.00),v40,z0,tPen\WObj:=wPaper;
    MoveL Offs(pOrigin,190.25,58.28,0.00),v40,z0,tPen\WObj:=wPaper;
    MoveL Offs(pOrigin,190.25,58.28,0.00),v40,z0,tPen\WObj:=wPaper;
    MoveL Offs(pOrigin,191.00,57.83,0.00),v40,z0,tPen\WObj:=wPaper;
    MoveL Offs(pOrigin,192.20,57.97,0.00),v40,z0,tPen\WObj:=wPaper;
    MoveL Offs(pOrigin,198.95,64.72,0.00),v40,z0,tPen\WObj:=wPaper;
    MoveL Offs(pOrigin,199.10,65.32,0.00),v40,z0,tPen\WObj:=wPaper;
    MoveL Offs(pOrigin,198.65,66.07,0.00),v40,fine,tPen\WObj:=wPaper;
    MoveL Offs(pOrigin,198.65,66.07,6.00),v60,z5,tPen\WObj:=wPaper;
    MoveL Offs(pOrigin,194.15,68.03,6.00),vTravel,z5,tPen\WObj:=wPaper;
    MoveL Offs(pOrigin,194.15,68.03,0.00),v60,z0,tPen\WObj:=wPaper;
    MoveL Offs(pOrigin,187.70,74.03,0.00),v40,fine,tPen\WObj:=wPaper;
    MoveL Offs(pOrigin,187.70,74.03,6.00),v60,z5,tPen\WObj:=wPaper;
    MoveL Offs(pOrigin,185.30,72.97,6.00),vTravel,z5,tPen\WObj:=wPaper;
    MoveL Offs(pOrigin,185.30,72.97,0.00),v60,z0,tPen\WObj:=wPaper;
    MoveL Offs(pOrigin,188.15,70.12,0.00),v40,z0,tPen\WObj:=wPaper;
    MoveL Offs(pOrigin,188.75,69.97,0.00),v40,z0,tPen\WObj:=wPaper;
    MoveL Offs(pOrigin,188.90,69.22,0.00),v40,z0,tPen\WObj:=wPaper;
    MoveL Offs(pOrigin,188.30,68.32,0.00),v40,fine,tPen\WObj:=wPaper;
    MoveL Offs(pOrigin,188.30,68.32,6.00),v60,z5,tPen\WObj:=wPaper;
    MoveL Offs(pOrigin,185.45,66.68,6.00),vTravel,z5,tPen\WObj:=wPaper;
    MoveL Offs(pOrigin,185.45,66.68,0.00),v60,z0,tPen\WObj:=wPaper;
    MoveL Offs(pOrigin,180.35,61.58,0.00),v40,z0,tPen\WObj:=wPaper;
    MoveL Offs(pOrigin,180.35,61.58,0.00),v40,z0,tPen\WObj:=wPaper;
    MoveL Offs(pOrigin,185.45,66.53,0.00),v40,z0,tPen\WObj:=wPaper;
    MoveL Offs(pOrigin,186.05,66.68,0.00),v40,z0,tPen\WObj:=wPaper;
    MoveL Offs(pOrigin,186.80,66.38,0.00),v40,z0,tPen\WObj:=wPaper;
    MoveL Offs(pOrigin,191.75,61.42,0.00),v40,fine,tPen\WObj:=wPaper;
    MoveL Offs(pOrigin,191.75,61.42,6.00),v60,z5,tPen\WObj:=wPaper;
    MoveL Offs(pOrigin,193.00,60.92,6.00),vTravel,z5,tPen\WObj:=wPaper;
    MoveL Offs(pOrigin,193.00,60.92,0.00),v60,z0,tPen\WObj:=wPaper;
    MoveL Offs(pOrigin,197.60,65.47,0.00),v40,z0,tPen\WObj:=wPaper;
    MoveL Offs(pOrigin,193.00,60.92,0.00),v40,fine,tPen\WObj:=wPaper;
    MoveL Offs(pOrigin,193.00,60.92,6.00),v60,z5,tPen\WObj:=wPaper;
    MoveL Offs(pOrigin,192.05,59.92,6.00),vTravel,z5,tPen\WObj:=wPaper;
    MoveL Offs(pOrigin,192.05,59.92,0.00),v60,z0,tPen\WObj:=wPaper;
    MoveL Offs(pOrigin,192.80,60.67,0.00),v40,z0,tPen\WObj:=wPaper;
    MoveL Offs(pOrigin,192.05,59.92,0.00),v40,fine,tPen\WObj:=wPaper;
    MoveL Offs(pOrigin,192.05,59.92,6.00),v60,z5,tPen\WObj:=wPaper;
    MoveL Offs(pOrigin,193.15,58.83,6.00),vTravel,z5,tPen\WObj:=wPaper;
    MoveL Offs(pOrigin,193.15,58.83,0.00),v60,z0,tPen\WObj:=wPaper;
    MoveL Offs(pOrigin,194.45,60.08,0.00),v40,z0,tPen\WObj:=wPaper;
    MoveL Offs(pOrigin,193.15,58.83,0.00),v40,z0,tPen\WObj:=wPaper;
    MoveL Offs(pOrigin,192.35,57.97,0.00),v40,z0,tPen\WObj:=wPaper;
    MoveL Offs(pOrigin,192.80,58.42,0.00),v40,z0,tPen\WObj:=wPaper;
    MoveL Offs(pOrigin,192.35,57.97,0.00),v40,fine,tPen\WObj:=wPaper;
    MoveL Offs(pOrigin,192.35,57.97,6.00),v60,z5,tPen\WObj:=wPaper;
    MoveL Offs(pOrigin,194.80,60.47,6.00),vTravel,z5,tPen\WObj:=wPaper;
    MoveL Offs(pOrigin,194.80,60.47,0.00),v60,z0,tPen\WObj:=wPaper;
    MoveL Offs(pOrigin,198.95,64.57,0.00),v40,z0,tPen\WObj:=wPaper;
    MoveL Offs(pOrigin,194.80,60.47,0.00),v40,fine,tPen\WObj:=wPaper;
    MoveL Offs(pOrigin,194.80,60.47,6.00),v60,z5,tPen\WObj:=wPaper;
    MoveL Offs(pOrigin,206.05,74.38,6.00),vTravel,z5,tPen\WObj:=wPaper;
    MoveL Offs(pOrigin,206.05,74.38,0.00),v60,z0,tPen\WObj:=wPaper;
    MoveL Offs(pOrigin,206.15,74.88,0.00),v40,z0,tPen\WObj:=wPaper;
    MoveL Offs(pOrigin,206.55,74.72,0.00),v40,z0,tPen\WObj:=wPaper;
    MoveL Offs(pOrigin,206.55,74.22,0.00),v40,z0,tPen\WObj:=wPaper;
    MoveL Offs(pOrigin,206.05,74.38,0.00),v40,fine,tPen\WObj:=wPaper;
    MoveL Offs(pOrigin,206.05,74.38,6.00),v60,z5,tPen\WObj:=wPaper;
    MoveL Offs(pOrigin,188.90,82.72,6.00),vTravel,z5,tPen\WObj:=wPaper;
    MoveL Offs(pOrigin,188.90,82.72,0.00),v60,z0,tPen\WObj:=wPaper;
    MoveL Offs(pOrigin,186.50,83.03,0.00),v40,fine,tPen\WObj:=wPaper;
    MoveL Offs(pOrigin,186.50,83.03,6.00),v60,z5,tPen\WObj:=wPaper;
    MoveL Offs(pOrigin,186.50,84.53,6.00),vTravel,z5,tPen\WObj:=wPaper;
    MoveL Offs(pOrigin,186.50,84.53,0.00),v60,z0,tPen\WObj:=wPaper;
    MoveL Offs(pOrigin,186.35,83.07,0.00),v40,z0,tPen\WObj:=wPaper;
    MoveL Offs(pOrigin,183.50,83.03,0.00),v40,z0,tPen\WObj:=wPaper;
    MoveL Offs(pOrigin,181.55,84.82,0.00),v40,z0,tPen\WObj:=wPaper;
    MoveL Offs(pOrigin,181.55,84.82,0.00),v40,z0,tPen\WObj:=wPaper;
    MoveL Offs(pOrigin,185.30,88.57,0.00),v40,z0,tPen\WObj:=wPaper;
    MoveL Offs(pOrigin,186.35,88.72,0.00),v40,z0,tPen\WObj:=wPaper;
    MoveL Offs(pOrigin,189.05,86.18,0.00),v40,fine,tPen\WObj:=wPaper;
    MoveL Offs(pOrigin,189.05,86.18,6.00),v60,z5,tPen\WObj:=wPaper;
    MoveL Offs(pOrigin,194.75,93.38,6.00),vTravel,z5,tPen\WObj:=wPaper;
    MoveL Offs(pOrigin,194.75,93.38,0.00),v60,z0,tPen\WObj:=wPaper;
    MoveL Offs(pOrigin,194.70,94.12,0.00),v40,z0,tPen\WObj:=wPaper;
    MoveL Offs(pOrigin,195.20,94.68,0.00),v40,z0,tPen\WObj:=wPaper;
    MoveL Offs(pOrigin,196.10,93.97,0.00),v40,z0,tPen\WObj:=wPaper;
    MoveL Offs(pOrigin,197.30,93.97,0.00),v40,z0,tPen\WObj:=wPaper;
    MoveL Offs(pOrigin,198.50,94.28,0.00),v40,z0,tPen\WObj:=wPaper;
    MoveL Offs(pOrigin,198.60,95.78,0.00),v40,z0,tPen\WObj:=wPaper;
    MoveL Offs(pOrigin,198.20,95.93,0.00),v40,z0,tPen\WObj:=wPaper;
    MoveL Offs(pOrigin,197.30,95.18,0.00),v40,z0,tPen\WObj:=wPaper;
    MoveL Offs(pOrigin,197.30,95.18,0.00),v40,z0,tPen\WObj:=wPaper;
    MoveL Offs(pOrigin,198.20,96.07,0.00),v40,z0,tPen\WObj:=wPaper;
    MoveL Offs(pOrigin,198.05,96.53,0.00),v40,z0,tPen\WObj:=wPaper;
    MoveL Offs(pOrigin,197.45,96.53,0.00),v40,z0,tPen\WObj:=wPaper;
    MoveL Offs(pOrigin,193.55,100.72,0.00),v40,fine,tPen\WObj:=wPaper;
    MoveL Offs(pOrigin,193.55,100.72,6.00),v60,z5,tPen\WObj:=wPaper;
    MoveL Offs(pOrigin,197.30,100.28,6.00),vTravel,z5,tPen\WObj:=wPaper;
    MoveL Offs(pOrigin,197.30,100.28,0.00),v60,z0,tPen\WObj:=wPaper;
    MoveL Offs(pOrigin,198.30,99.07,0.00),v40,z0,tPen\WObj:=wPaper;
    MoveL Offs(pOrigin,198.95,97.12,0.00),v40,z0,tPen\WObj:=wPaper;
    MoveL Offs(pOrigin,198.80,96.68,0.00),v40,fine,tPen\WObj:=wPaper;
    MoveL Offs(pOrigin,198.80,96.68,6.00),v60,z5,tPen\WObj:=wPaper;
    MoveL Offs(pOrigin,197.30,100.28,6.00),vTravel,z5,tPen\WObj:=wPaper;
    MoveL Offs(pOrigin,197.30,100.28,0.00),v60,z0,tPen\WObj:=wPaper;
    MoveL Offs(pOrigin,198.95,101.93,0.00),v40,fine,tPen\WObj:=wPaper;
    MoveL Offs(pOrigin,198.95,101.93,6.00),v60,z5,tPen\WObj:=wPaper;
    MoveL Offs(pOrigin,203.45,112.57,6.00),vTravel,z5,tPen\WObj:=wPaper;
    MoveL Offs(pOrigin,203.45,112.57,0.00),v60,z0,tPen\WObj:=wPaper;
    MoveL Offs(pOrigin,211.70,104.03,0.00),v40,fine,tPen\WObj:=wPaper;
    MoveL Offs(pOrigin,211.70,104.03,6.00),v60,z5,tPen\WObj:=wPaper;
    MoveL Offs(pOrigin,210.80,101.78,6.00),vTravel,z5,tPen\WObj:=wPaper;
    MoveL Offs(pOrigin,210.80,101.78,0.00),v60,z0,tPen\WObj:=wPaper;
    MoveL Offs(pOrigin,202.60,109.72,0.00),v40,z0,tPen\WObj:=wPaper;
    MoveL Offs(pOrigin,202.55,110.62,0.00),v40,z0,tPen\WObj:=wPaper;
    MoveL Offs(pOrigin,203.45,112.57,0.00),v40,fine,tPen\WObj:=wPaper;
    MoveL Offs(pOrigin,203.45,112.57,6.00),v60,z5,tPen\WObj:=wPaper;
    MoveL Offs(pOrigin,204.35,115.28,6.00),vTravel,z5,tPen\WObj:=wPaper;
    MoveL Offs(pOrigin,204.35,115.28,0.00),v60,z0,tPen\WObj:=wPaper;
    MoveL Offs(pOrigin,206.75,113.32,0.00),v40,z0,tPen\WObj:=wPaper;
    MoveL Offs(pOrigin,207.05,113.18,0.00),v40,z0,tPen\WObj:=wPaper;
    MoveL Offs(pOrigin,212.75,107.18,0.00),v40,fine,tPen\WObj:=wPaper;
    MoveL Offs(pOrigin,212.75,107.18,6.00),v60,z5,tPen\WObj:=wPaper;
    MoveL Offs(pOrigin,213.65,108.07,6.00),vTravel,z5,tPen\WObj:=wPaper;
    MoveL Offs(pOrigin,213.65,108.07,0.00),v60,z0,tPen\WObj:=wPaper;
  ENDPROC

  PROC DrawPart17()
    MoveL Offs(pOrigin,204.95,116.93,0.00),v40,z0,tPen\WObj:=wPaper;
    MoveL Offs(pOrigin,204.90,117.53,0.00),v40,z0,tPen\WObj:=wPaper;
    MoveL Offs(pOrigin,205.55,118.28,0.00),v40,z0,tPen\WObj:=wPaper;
    MoveL Offs(pOrigin,205.55,118.28,0.00),v40,z0,tPen\WObj:=wPaper;
    MoveL Offs(pOrigin,205.55,119.47,0.00),v40,z0,tPen\WObj:=wPaper;
    MoveL Offs(pOrigin,206.00,119.93,0.00),v40,z0,tPen\WObj:=wPaper;
    MoveL Offs(pOrigin,206.00,120.22,0.00),v40,z0,tPen\WObj:=wPaper;
    MoveL Offs(pOrigin,210.20,115.68,0.00),v40,z0,tPen\WObj:=wPaper;
    MoveL Offs(pOrigin,215.75,121.43,0.00),v40,z0,tPen\WObj:=wPaper;
    MoveL Offs(pOrigin,215.30,122.18,0.00),v40,z0,tPen\WObj:=wPaper;
    MoveL Offs(pOrigin,209.30,123.82,0.00),v40,z0,tPen\WObj:=wPaper;
    MoveL Offs(pOrigin,206.15,120.82,0.00),v40,z0,tPen\WObj:=wPaper;
    MoveL Offs(pOrigin,206.00,120.22,0.00),v40,fine,tPen\WObj:=wPaper;
    MoveL Offs(pOrigin,206.00,120.22,6.00),v60,z5,tPen\WObj:=wPaper;
    MoveL Offs(pOrigin,207.20,122.03,6.00),vTravel,z5,tPen\WObj:=wPaper;
    MoveL Offs(pOrigin,207.20,122.03,0.00),v60,z0,tPen\WObj:=wPaper;
    MoveL Offs(pOrigin,208.70,123.53,0.00),v40,z0,tPen\WObj:=wPaper;
    MoveL Offs(pOrigin,207.20,122.03,0.00),v40,fine,tPen\WObj:=wPaper;
    MoveL Offs(pOrigin,207.20,122.03,6.00),v60,z5,tPen\WObj:=wPaper;
    MoveL Offs(pOrigin,190.25,121.43,6.00),vTravel,z5,tPen\WObj:=wPaper;
    MoveL Offs(pOrigin,190.25,121.43,0.00),v60,z0,tPen\WObj:=wPaper;
    MoveL Offs(pOrigin,185.00,116.18,0.00),v40,fine,tPen\WObj:=wPaper;
    MoveL Offs(pOrigin,185.00,116.18,6.00),v60,z5,tPen\WObj:=wPaper;
    MoveL Offs(pOrigin,183.50,114.82,6.00),vTravel,z5,tPen\WObj:=wPaper;
    MoveL Offs(pOrigin,183.50,114.82,0.00),v60,z0,tPen\WObj:=wPaper;
    MoveL Offs(pOrigin,184.25,115.57,0.00),v40,z0,tPen\WObj:=wPaper;
    MoveL Offs(pOrigin,183.50,114.82,0.00),v40,fine,tPen\WObj:=wPaper;
    MoveL Offs(pOrigin,183.50,114.82,6.00),v60,z5,tPen\WObj:=wPaper;
    MoveL Offs(pOrigin,187.55,112.12,6.00),vTravel,z5,tPen\WObj:=wPaper;
    MoveL Offs(pOrigin,187.55,112.12,0.00),v60,z0,tPen\WObj:=wPaper;
    MoveL Offs(pOrigin,188.25,112.72,0.00),v40,z0,tPen\WObj:=wPaper;
    MoveL Offs(pOrigin,189.80,116.93,0.00),v40,fine,tPen\WObj:=wPaper;
    MoveL Offs(pOrigin,189.80,116.93,6.00),v60,z5,tPen\WObj:=wPaper;
    MoveL Offs(pOrigin,181.00,123.32,6.00),vTravel,z5,tPen\WObj:=wPaper;
    MoveL Offs(pOrigin,181.00,123.32,0.00),v60,z0,tPen\WObj:=wPaper;
    MoveL Offs(pOrigin,182.30,124.57,0.00),v40,z0,tPen\WObj:=wPaper;
    MoveL Offs(pOrigin,181.00,123.32,0.00),v40,fine,tPen\WObj:=wPaper;
    MoveL Offs(pOrigin,181.00,123.32,6.00),v60,z5,tPen\WObj:=wPaper;
    MoveL Offs(pOrigin,179.60,121.88,6.00),vTravel,z5,tPen\WObj:=wPaper;
    MoveL Offs(pOrigin,179.60,121.88,0.00),v60,z0,tPen\WObj:=wPaper;
    MoveL Offs(pOrigin,180.80,123.07,0.00),v40,z0,tPen\WObj:=wPaper;
    MoveL Offs(pOrigin,179.60,121.88,0.00),v40,fine,tPen\WObj:=wPaper;
    MoveL Offs(pOrigin,179.60,121.88,6.00),v60,z5,tPen\WObj:=wPaper;
    MoveL Offs(pOrigin,210.50,100.12,6.00),vTravel,z5,tPen\WObj:=wPaper;
    MoveL Offs(pOrigin,210.50,100.12,0.00),v60,z0,tPen\WObj:=wPaper;
    MoveL Offs(pOrigin,210.20,99.68,0.00),v40,z0,tPen\WObj:=wPaper;
    MoveL Offs(pOrigin,210.20,97.72,0.00),v40,z0,tPen\WObj:=wPaper;
    MoveL Offs(pOrigin,210.20,98.03,0.00),v40,fine,tPen\WObj:=wPaper;
    MoveL Offs(pOrigin,210.20,98.03,6.00),v60,z5,tPen\WObj:=wPaper;
    MoveL Offs(pOrigin,20.15,52.42,6.00),vTravel,z5,tPen\WObj:=wPaper;
    MoveL Offs(pOrigin,20.15,52.42,0.00),v60,z0,tPen\WObj:=wPaper;
    MoveL Offs(pOrigin,20.60,52.72,0.00),v40,z0,tPen\WObj:=wPaper;
    MoveL Offs(pOrigin,20.15,52.42,0.00),v40,fine,tPen\WObj:=wPaper;
    MoveL Offs(pOrigin,20.15,52.42,6.00),v60,z5,tPen\WObj:=wPaper;
  ENDPROC

ENDMODULE
